Yaskawa INFORM job: SKRZYNIA_5040_0_STOPNI_1OBR.JBI

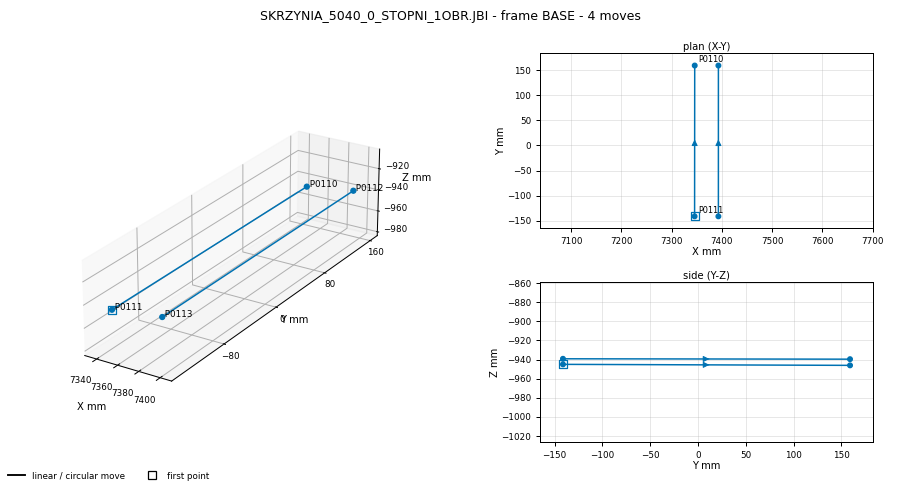
[picture p0: tool path of SKRZYNIA_5040_0_STOPNI_1OBR.JBI in frame BASE, 4 of 438 moves have a stored position in this frame; points joined in program order, loops and branches not executed]
/JOB
//NAME SKRZYNIA_5040_0_STOPNI_1OBR
///FOLDERNAME 02-SKRZYNIE_JOBS
//POS
///NPOS 514,514,0,47,4,0
///TOOL 0
///POSTYPE PULSE
///PULSE
C00000=1055,-24125,84372,288,19725,204
C00001=1055,-24125,84372,288,19725,204
C00002=25524,-25821,36823,19654,-58495,38520
C00003=23988,-24960,37134,18595,-57837,38812
C00004=22822,-23954,37534,17811,-57199,39017
C00005=22935,-24057,37491,17887,-57262,38997
C00006=20006,-24258,37408,15644,-56932,39751
C00007=24402,-25289,37013,18874,-58060,38740
C00008=22585,-24665,40358,17164,-59622,30036
C00009=23477,-23257,40205,18030,-58646,29630
C00010=22519,-22398,40568,17384,-58125,29795
C00011=22700,-22567,40495,17506,-58225,29764
C00012=19339,-22794,40398,14955,-57865,30607
C00013=24825,-24328,39798,18931,-59350,29401
C00014=0,-15438,65714,0,-68532,0
C00015=25524,-25821,36823,19654,-58495,38520
C00016=23988,-24960,37134,18595,-57837,38812
C00017=22822,-23954,37534,17811,-57199,39017
C00018=22935,-24057,37491,17887,-57262,38997
C00019=20006,-24258,37408,15644,-56932,39751
C00020=24402,-25289,37013,18874,-58060,38740
C00021=22585,-24665,40358,17164,-59622,30036
C00022=23477,-23257,40205,18030,-58646,29630
C00023=22519,-22398,40568,17384,-58125,29795
C00024=22700,-22567,40495,17506,-58225,29764
C00025=19339,-22794,40398,14955,-57865,30607
C00026=24825,-24328,39798,18931,-59350,29401
C00027=32755,-32613,25711,29640,-48730,33694
C00028=25632,-30899,26166,23992,-46203,35378
C00029=24264,-29862,26497,22996,-45413,35639
C00030=24403,-29974,26459,23097,-45496,35612
C00031=20575,-30233,26374,19602,-44891,36810
C00032=26556,-31526,25988,24663,-46720,35206
C00033=30846,-32795,25752,28021,-48338,30427
C00034=24953,-30697,26306,23444,-45946,31743
C00035=23937,-29910,26558,22702,-45353,31936
C00036=24039,-29993,26530,22778,-45414,31916
C00037=20322,-30240,26449,19379,-44834,33080
C00038=25997,-31433,26093,24205,-46535,31545
C00039=26028,-43665,26580,-39946,8682,24640
C00040=27956,-30595,53065,-101898,6609,54413
C00041=26028,-43663,26580,-39944,8677,24639
C00042=38784,-34544,25404,33956,-51320,34445
C00043=29266,-32676,25756,26732,-47889,36488
C00044=25734,-31262,26119,24020,-46377,37252
C00045=24289,-30200,26441,22967,-45549,37525
C00046=24367,-30262,26420,23025,-45594,37511
C00047=20043,-30544,26331,19080,-44922,38860
C00048=26573,-31816,25967,24631,-46839,37095
C00049=27817,-32566,25782,25532,-47502,36865
C00050=26896,-32020,25916,24865,-47014,37034
C00051=24344,-30243,26427,23007,-45578,37515
C00052=24432,-30312,26405,23072,-45630,37498
C00053=20021,-30599,26315,19050,-44944,38872
C00054=26262,-31616,26021,24405,-46667,37153
C00055=27439,-32346,25835,25259,-47302,36935
C00056=27343,-32252,25856,25196,-47233,36946
C00057=24581,-30384,26384,23190,-45695,37464
C00058=24689,-30466,26358,23269,-45758,37444
C00059=20001,-30771,26264,18999,-45026,38899
C00060=26308,-31607,26026,24448,-46671,37139
C00061=27526,-32360,25834,25329,-47326,36914
C00062=24269,-40076,6479,29767,-34177,34232
C00063=22958,-37632,10123,27061,-35370,35326
C00064=22703,-41294,1722,31272,-29953,33282
C00065=19440,-41515,1663,27208,-29122,34832
C00066=25465,-43501,1200,33269,-31905,32752
C00067=87177,-39066,-1236,81808,-72661,19198
C00068=4794,-34097,38974,4189,-31824,-1302
C00069=4794,-34097,38974,4189,13412,-1302
C00070=5394,-34032,37825,4779,8346,-1512
C00071=6591,-33902,35532,5956,-1761,-1932
C00072=10065,-33530,28876,9373,-31104,-3154
C00073=31877,-32319,25770,29025,-48287,33360
C00074=25247,-31158,26079,23631,-46177,35016
C00075=23652,-29939,26460,22464,-45250,35320
C00076=23742,-30013,26436,22530,-45305,35302
C00077=19630,-30281,26348,18756,-44677,36597
C00078=26056,-31710,25928,24219,-46631,34863
C00079=38095,-40136,7813,41252,-44156,24924
C00080=33231,-38681,8176,37792,-41757,25918
C00081=31538,-37640,8473,36716,-40716,26179
C00082=31687,-37737,8444,36811,-40809,26155
C00083=27389,-38154,8322,32773,-39589,27627
C00084=33834,-39023,8084,38175,-42120,25821
C00085=4264,-34194,25387,4006,-26954,-29436
C00086=4264,-34194,25387,4006,-26954,-81856
C00087=17634,-23800,39238,9573,-31425,-73339
C00088=17837,-27228,32238,10495,-29236,-73805
C00089=17837,-21535,44509,9322,-33342,-73155
C00090=17548,-20734,45666,8935,-33511,-73021
C00091=-20829,-18800,50532,-12466,-37179,-77446
C00092=-20884,-20901,46110,-12960,-35762,-77182
C00093=-20884,-26676,33664,-14451,-31668,-76336
C00094=-20624,-26699,33167,-14265,-31320,-76369
C00095=-33629,-40566,17444,-29603,-33447,-71192
C00096=-33629,-40566,17444,42578,-32312,-84654
C00097=-42160,-31266,16400,42578,-32312,-84654
C00098=-87798,-804,48829,-20188,-26072,-60966
C00099=-76454,-11934,10236,-25964,7954,-64922
C00100=-76448,-11928,10235,-25961,7944,-64914
C00101=-68643,-7759,-23318,-14097,50582,-74897
C00102=-70868,-8793,-8075,-29663,30364,-70765
C00103=-67243,-1968,12282,-49553,26687,-63567
C00104=-68655,-309,14069,-48513,25966,-64203
C00105=-67497,-1678,12591,-49367,26558,-63682
C00106=-71436,-723,2905,-26484,35140,-73726
C00107=-71436,176,6426,-27636,33595,-73066
C00108=-71434,778,8668,-28412,32633,-72624
C00109=-68624,-2689,-85,-28291,36551,-72622
C00110=-99375,3692,5712,40719,48607,-84097
C00111=-94964,4957,10918,40408,44640,-83792
C00112=-93063,6047,12199,39572,43744,-83178
C00113=-94964,4957,10918,40408,44640,-83792
C00114=-94964,5754,13918,41385,43553,-84439
C00115=-94964,4957,10918,40408,44640,-83792
C00116=-90271,-412,-5146,23417,46876,-76529
C00117=-83133,-4088,-8267,6704,41492,-71542
C00118=-83133,-4088,-8267,6704,41492,-71542
C00119=-83133,-4088,-8267,6704,41492,-11598
C00120=-83133,-16026,-8267,6704,41492,-11598
C00121=-83133,-16026,-8267,6704,41492,-11598
C00122=-48225,-19387,30619,3889,32460,-6728
C00123=56943,-39861,25115,1795,-37402,-69601
C00124=29960,-38386,-19607,-115769,-41858,-24264
C00125=65721,-6478,18155,-133323,-22195,3361
C00126=70544,4411,32968,-134868,-18623,4660
C00127=71874,8263,38598,-134556,-17327,4659
C00128=72629,9390,40002,-135279,-16924,5107
C00129=71441,7638,37831,-134139,-17555,4406
C00130=77146,8888,25050,-166574,-32612,18372
C00131=77146,10029,28643,-166204,-31014,18167
C00132=77146,11198,32202,-165803,-29459,17947
C00133=75508,4678,16951,-165715,-35157,17778
C00134=68680,12216,24468,-164340,-40455,-13359
C00135=68362,12845,25743,-164045,-40097,-13561
C00136=68362,13700,28585,-163752,-38808,-13742
C00137=68362,12845,25743,-164045,-40097,-13561
C00138=64993,-1168,28876,-102971,-10760,-49875
C00139=63888,481,30670,-102324,-11438,-50313
C00140=64993,-1168,28876,-102971,-10760,-49875
C00141=58588,-14653,4620,-120782,-19611,-35794
C00142=29960,-38386,-19607,-115769,-41858,-24264
C00143=56943,-39861,25115,1795,-37402,-69601
C00144=-1002,-39861,25115,1795,-37402,-69601
C00145=-1001,-39858,25114,1795,-37402,0
C00146=6591,-33902,35532,5956,-1761,-1932
C00147=6592,-33900,35531,103508,-35512,-26314
C00148=-99253,-13690,44082,59847,13407,-31313
C00149=-85045,-36869,-4353,28502,-22832,-52282
C00150=-92346,-18713,13565,21110,-22545,-55257
C00151=-85370,-14218,16934,32905,-23649,-60330
C00152=-84150,-13282,17685,34842,-23935,-61163
C00153=-82877,-12536,18624,36445,-24482,-61818
C00154=-84150,-13282,17685,34842,-23935,-61163
C00155=-85467,-11480,19558,33086,-23405,-60436
C00156=-84150,-13282,17685,34842,-23935,-61163
C00157=-85732,-21202,11427,30682,-24763,-59235
C00158=-84559,-15616,15722,33768,-24118,-60665
C00159=-84150,-13282,17685,34842,-23935,-61163
C00160=-83260,-12880,18034,36130,-24218,-61709
C00161=-84150,-13282,17685,34842,-23935,-61163
C00162=-85365,-11775,19006,33430,-23307,-60600
C00163=-84150,-13282,17685,34842,-23935,-61163
C00164=-85786,-16909,14677,31743,-23900,-59790
C00165=-84150,-13282,17685,34842,-23935,-61163
C00166=-83215,-12861,18051,36194,-24233,-61735
C00167=-84150,-13282,17685,34842,-23935,-61163
C00168=-85327,-11825,18959,33476,-23327,-60618
C00169=-84150,-13282,17685,34842,-23935,-61163
C00170=-87841,-18519,13420,28367,-23534,-58339
C00171=-84150,-13282,17685,34842,-23935,-61163
C00172=-83292,-12894,18020,36083,-24208,-61688
C00173=-84150,-13282,17685,34842,-23935,-61163
C00174=-85185,-12008,18799,33646,-23400,-60687
C00175=-84150,-13282,17685,34842,-23935,-61163
C00176=-86371,-18277,13606,30568,-23951,-59265
C00177=-84345,-13370,17612,34554,-23873,-61041
C00178=-83240,-12871,18042,36158,-24225,-61720
C00179=-84345,-13370,17612,34554,-23873,-61041
C00180=-85365,-12110,18711,33368,-23345,-60568
C00181=-84345,-13370,17612,34554,-23873,-61041
C00182=-86191,-19647,12567,30467,-24278,-59187
C00183=-84345,-13372,17610,34552,-23873,-61039
C00184=-83096,-12807,18098,36363,-24268,-61804
C00185=-84345,-13372,17610,34552,-23873,-61039
C00186=-85268,-12232,18600,33480,-23393,-60612
C00187=-84345,-13372,17610,34552,-23873,-61039
C00188=-84814,-16043,15376,33312,-24093,-60464
C00189=-84104,-13265,17702,34906,-23948,-61189
C00190=-82960,-12743,18153,36555,-24313,-61887
C00191=-84104,-13265,17702,34906,-23948,-61189
C00192=-84979,-12194,18635,33901,-23496,-60788
C00193=-84104,-13265,17702,34906,-23948,-61189
C00194=-86610,-16845,14732,30573,-23614,-59301
C00195=-84104,-13265,17702,34906,-23948,-61189
C00196=-82793,-12667,18222,36790,-24370,-61986
C00197=-84104,-13265,17702,34906,-23948,-61189
C00198=-84888,-12305,18537,34004,-23540,-60830
C00199=-84104,-13265,17702,34906,-23948,-61189
C00200=-83806,-19585,12613,33764,-25080,-60559
C00201=-83675,-13072,17868,35530,-24083,-61453
C00202=-82553,-12556,18319,37130,-24451,-62127
C00203=-83675,-13072,17868,35530,-24083,-61453
C00204=-84378,-12223,18610,34735,-23716,-61138
C00205=-83675,-13072,17868,35530,-24083,-61453
C00206=-87149,-17993,13826,29513,-23647,-58830
C00207=-84104,-13265,17702,34906,-23948,-61189
C00208=-82640,-12594,18285,37014,-24425,-62079
C00209=-84104,-13265,17702,34906,-23948,-61189
C00210=-84792,-12429,18430,34119,-23592,-60877
C00211=-84104,-13265,17702,34906,-23948,-61189
C00212=-83583,-9185,30892,23668,-36042,-57025
C00213=-85789,-8328,35795,20592,-37093,-55378
C00214=-85786,-16735,14816,31782,-23869,-59812
C00215=-84103,-13263,17702,34906,-23947,-61191
C00216=-83225,-12865,18046,36177,-24227,-61729
C00217=-84103,-13263,17702,34906,-23947,-61191
C00218=-84774,-12447,18412,34138,-23599,-60886
C00219=-84103,-13263,17702,34906,-23947,-61191
C00220=-86149,-16246,6730,18897,-35239,-57128
C00221=-86244,-15289,7532,18875,-35060,-57127
C00222=-85361,-14893,7870,19824,-35193,-57574
C00223=-86244,-15289,7532,18875,-35060,-57127
C00224=-86889,-14409,8282,18264,-34784,-56850
C00225=-86244,-15289,7532,18875,-35060,-57127
C00226=-90262,-21765,2389,14114,-35574,-54847
C00227=-90262,-21765,2389,28730,-17672,-54847
C00228=-89967,-19086,25635,28730,-17672,-54847
C00229=568,-24029,84339,168,19981,112
C00230=568,-24677,83015,164,20405,113
C00231=101153,-24598,83176,165,20353,113
C00232=101153,-24598,83176,165,20353,113
C00233=89967,-19086,25635,-28730,-17672,54847
C00234=90262,-21765,2389,-28730,-17672,54847
C00235=86932,-18662,4771,-17876,-35519,56628
C00236=86578,-15436,7408,-18515,-35011,56957
C00237=85428,-14922,7844,-19753,-35183,57541
C00238=84405,-14447,8250,-20842,-35348,58054
C00239=85428,-14922,7844,-19753,-35183,57541
C00240=86134,-13973,8661,-19091,-34881,57237
C00241=85428,-14922,7844,-19753,-35183,57541
C00242=85786,-16735,14816,-31782,-23869,59812
C00243=83514,-12996,17929,-35760,-24132,61552
C00244=82296,-12429,18424,-37488,-24534,62281
C00245=83514,-12996,17929,-35760,-24132,61552
C00246=84266,-12085,18725,-34910,-23738,61214
C00247=83514,-12996,17929,-35760,-24132,61552
C00248=87323,-6914,39851,-18853,-38149,44508
C00249=83118,-12818,18089,-36330,-24263,61791
C00250=81969,-12276,18566,-37944,-24648,62472
C00251=83118,-12818,18089,-36330,-24263,61791
C00252=83927,-11846,18941,-35423,-23842,61433
C00253=83118,-12818,18089,-36330,-24263,61791
C00254=83806,-19585,12613,-33764,-25080,60559
C00255=83148,-12832,18077,-36287,-24254,61773
C00256=81889,-12236,18598,-38058,-24676,62520
C00257=83148,-12832,18077,-36287,-24254,61773
C00258=83900,-11930,18867,-35446,-23862,61440
C00259=83148,-12832,18077,-36287,-24254,61773
C00260=86610,-16845,14732,-30573,-23614,59301
C00261=82493,-13239,17725,-37070,-24559,62089
C00262=81442,-12739,18159,-38529,-24915,62703
C00263=82493,-13239,17725,-37070,-24559,62089
C00264=83435,-12133,18689,-36040,-24063,61682
C00265=82493,-13239,17725,-37070,-24559,62089
C00266=84814,-16043,15376,-33312,-24093,60464
C00267=82555,-13613,17404,-36910,-24580,62015
C00268=81369,-13053,17885,-38558,-24979,62709
C00269=82555,-13613,17404,-36910,-24580,62015
C00270=83568,-12431,18429,-35805,-24046,61580
C00271=82555,-13613,17404,-36910,-24580,62015
C00272=86191,-19647,12567,-30467,-24278,59187
C00273=82500,-13648,17375,-36975,-24607,62039
C00274=81594,-13224,17740,-38236,-24911,62571
C00275=82500,-13648,17375,-36975,-24607,62039
C00276=83449,-12543,18332,-35941,-24104,61633
C00277=82500,-13648,17375,-36975,-24607,62039
C00278=86371,-18277,13606,-30568,-23951,59265
C00279=82904,-13790,17251,-36416,-24470,61808
C00280=81796,-13275,17692,-37971,-24838,62464
C00281=82904,-13790,17251,-36416,-24470,61808
C00282=83696,-12867,18046,-35547,-24051,61466
C00283=82904,-13790,17251,-36416,-24470,61808
C00284=87841,-18519,13420,-28367,-23534,58339
C00285=82748,-13879,17174,-36603,-24542,61883
C00286=81789,-13434,17554,-37946,-24861,62449
C00287=82748,-13879,17174,-36603,-24542,61883
C00288=83603,-12888,18026,-35668,-24086,61514
C00289=82748,-13879,17174,-36603,-24542,61883
C00290=85786,-16909,14677,-31743,-23900,59790
C00291=82339,-14116,16972,-37087,-24733,62079
C00292=81557,-13752,17280,-38171,-24994,62536
C00293=82339,-14116,16972,-37087,-24733,62079
C00294=83390,-12909,18006,-35951,-24172,61633
C00295=82339,-14116,16972,-37087,-24733,62079
C00296=85732,-21202,11427,-30682,-24763,59235
C00297=82398,-14365,16763,-36952,-24745,62014
C00298=81340,-13876,17176,-38416,-25096,62632
C00299=82398,-14365,16763,-36952,-24745,62014
C00300=83629,-12951,17972,-35620,-24090,61491
C00301=82398,-14365,16763,-36952,-24745,62014
C00302=92346,-18713,13565,-21110,-22545,55257
C00303=82794,-13980,17083,-36511,-24538,61844
C00304=81697,-13472,17516,-38043,-24902,62488
C00305=82794,-13980,17083,-36511,-24538,61844
C00306=83767,-12847,18056,-35444,-24023,61424
C00307=82794,-13980,17083,-36511,-24538,61844
C00308=85045,-36869,-4353,-28502,-22832,52282
C00309=69856,-53931,-13446,-33557,-28911,29591
C00310=73943,-28815,39553,-16801,-45089,19004
C00311=0,-24029,84339,0,19981,0
C00312=0,-24029,84339,0,19981,0
C00313=0,-52280,40443,0,6876,0
C00314=63961,-36661,14391,66570,-58199,13439
C00315=49610,-38907,493,64064,-47684,11073
C00316=46884,-37851,878,62974,-45995,11189
C00317=46721,-37909,857,62857,-45922,11231
C00318=54160,-39955,137,66075,-50361,10746
C00319=0,-52280,40443,0,6876,0
C00320=0,-52280,40443,0,6876,0
C00321=42978,-45587,7631,48214,-41849,18034
C00322=36694,-44945,-1657,49443,-34807,15750
C00323=45435,-38965,-3578,70378,-41546,11426
C00324=45248,-39111,-3491,69948,-41437,11613
C00325=32579,-45219,-13334,65473,-28542,22073
C00326=59828,-44646,-5405,72855,-48572,12139
C00327=0,-38761,66314,0,-763,0
C00328=0,-44757,54667,0,2744,0
C00329=40382,-38226,12225,48505,-40693,16039
C00330=55481,-27484,23768,62968,-54833,11978
C00331=49777,-26559,24206,59885,-51900,12566
C00332=49523,-31326,12270,55024,-55929,13117
C00333=55330,-33748,11238,57660,-59334,12681
C00334=78664,-24436,10378,82837,-79111,12029
C00335=75189,-23065,11287,81851,-76948,11927
C00336=75189,-45249,11287,81851,-38847,11927
C00337=29880,-45249,11287,43145,-11324,11927
C00338=0,-24029,84339,0,19981,0
C00339=0,-24026,84338,1,19977,2
C00340=4264,-34194,25387,4006,-26954,-29436
C00341=4264,-34194,25387,4006,-26954,-81856
C00342=18580,-28601,30698,11472,-29284,-74138
C00343=-23778,-26243,38799,-16502,-35132,-75964
C00344=18580,-28601,30698,11472,-29284,-74138
C00345=4264,-34194,25387,4006,-26954,-81856
C00346=4264,-34194,25387,4006,-26954,-29436
C00347=1,-24024,84337,2,19973,1
C00348=-64243,-26178,31107,-39513,40312,-5844
C00349=-72148,3973,56008,-35470,42045,-10522
C00350=-72090,16396,76301,-42067,35650,-6519
C00351=-69388,15725,61378,-31740,35177,-8719
C00352=-69127,27099,75569,-32744,34250,-8088
C00353=-67573,2495,11285,-21767,57629,-15193
C00354=-77819,19629,29798,-10454,63174,-20704
C00355=-72990,23583,14304,-10735,77209,-20379
C00356=-74593,38003,46707,-11043,65751,-19814
C00357=-73236,38943,48295,-11400,65557,-19316
C00358=-73329,42107,51779,-6346,67443,-19636
C00359=-87142,34654,46174,17622,63862,-25393
C00360=-87240,36727,48611,18897,66604,-25032
C00361=-99033,21517,12213,24947,79702,-26203
C00362=-91500,-14196,-34781,24472,81625,-22832
C00363=-100472,-45007,-27818,8167,67201,-29302
C00364=0,-36642,16905,0,48372,0
C00365=66009,-61997,-62105,21406,63483,18379
C00366=97242,-23579,-39442,10179,68876,30321
C00367=73684,-7073,-17511,24638,68131,29022
C00368=59136,7235,6676,33270,66602,27507
C00369=54816,14937,6234,39741,69494,31070
C00370=54365,20668,19279,41017,66202,29418
C00371=64503,4223,2857,29650,48528,26647
C00372=75622,3202,-3149,3890,49494,34281
C00373=88036,13177,2413,-18568,66573,35876
C00374=90462,21593,10123,-22613,76266,34479
C00375=92450,29224,20002,-25750,81642,33727
C00376=94949,8131,-12163,-20291,74229,36861
C00377=94949,8084,-13484,-20215,75047,36712
C00378=70412,-34016,-52305,-11724,65624,29757
C00379=44268,-30306,-1568,-7370,48673,18708
C00380=1,-24024,84337,2,19973,1
C00381=1,-24024,84337,2,19973,1
C00382=3796,-57671,22373,2336,-25309,-753
C00383=52632,-34554,16626,51161,-63050,5622
C00384=59461,-32779,9832,66317,-58406,17312
C00385=52772,-27880,19104,60329,-56577,14845
C00386=51509,-17404,41655,51674,-64690,19351
C00387=62932,-33588,12189,66848,-61063,18031
C00388=55769,-31640,17107,64026,-54372,11197
C00389=50117,-26891,23585,59871,-52280,12556
C00390=49716,-31387,12242,55119,-56039,13097
C00391=55330,-33748,11238,57660,-59334,12681
C00392=1,-24024,84337,2,19973,1
C00393=1,-24024,84337,2,19973,1
C00394=57188,-41777,19973,48132,-58706,4905
C00395=55566,-48748,-16991,79805,-45048,-6941
C00396=49908,-48716,-25784,90749,-41340,-3650
C00397=43896,-46926,-25352,90956,-37526,-4581
C00398=43530,-46832,-25319,90960,-37294,-4630
C00399=55479,-50244,-26473,91085,-44870,-3042
C00400=12119,-24859,71505,13236,4440,2633
C00401=-91085,-34291,10385,1908,-24348,-42097
C00402=-86191,-19647,12567,30467,-24278,-59187
C00403=-99288,-11708,19065,-14233,-20220,-40075
C00404=-98206,-11518,19604,-10142,-20308,-41629
C00405=-99474,-20389,12397,-11593,-22150,-41069
C00406=0,-52280,40443,0,6876,0
C00407=85348,-24204,23536,-13963,-15515,44275
C00408=84670,-17015,14597,-33277,-24304,60423
C00409=96971,-12584,18294,8365,-19955,42614
C00410=97182,-12918,18001,8747,-20027,42449
C00411=96230,-24528,9149,6144,-22576,43630
C00412=0,-52280,40443,0,6876,0
C00413=0,-52280,40443,0,6876,0
C00414=-90140,-60305,18108,-2708,1721,-7625
C00415=-95594,-27428,6866,-4663,-19832,-42154
C00416=-99356,-13410,18355,-15385,-17730,-37479
C00417=-99405,-10878,20508,-15853,-17333,-37255
C00418=-99132,-10804,20575,-15274,-17279,-37502
C00419=-99132,-3482,39129,-10940,-24351,-39674
C00420=-97546,-6584,14255,-163983,-14128,32873
C00421=-100183,-18601,14070,-16273,-18800,-37146
C00422=-90140,-60305,18108,-2708,1721,-7625
C00423=0,-52280,40443,0,6876,0
C00424=84259,-57935,27522,-3761,3673,6310
C00425=86507,-39672,4297,-27618,-16640,46340
C00426=70477,-27878,7073,-45786,-32339,64941
C00427=84043,-16293,15174,-34312,-24409,60872
C00428=100395,-12639,18246,19464,-20904,37830
C00429=99154,-17369,4403,32227,-9753,28926
C00430=99154,-17369,4403,32227,-9753,28926
C00431=98497,-14262,-10338,-9662,27059,46922
C00432=97745,-17327,14348,11122,-20983,41455
C00433=86507,-39672,4297,-27618,-16640,46340
C00434=84259,-57935,27522,-3761,3673,6310
C00435=0,-52280,40443,0,6876,0
C00436=0,-27933,77061,0,20812,0
C00437=0,-27933,77061,0,20812,0
C00438=0,-52280,40443,0,6876,0
C00439=-91970,-60791,14435,-3343,512,-9412
C00440=-99196,-15868,16098,-13748,-19297,-38710
C00441=-99196,-15868,16098,-13748,-19297,-38710
C00442=-99196,-15868,16098,-13748,-19297,-38710
C00443=-85815,-11758,19597,31748,-21097,-58265
C00444=-87383,-11883,19487,26986,-20206,-56250
C00445=-99562,-16264,15781,-14410,-19427,-38431
C00446=-99196,-15868,16098,-13748,-19297,-38710
C00447=-91970,-60791,14435,-3343,512,-9412
C00448=0,-52280,40443,0,6876,0
C00449=91083,-60784,14823,-9043,-825,15173
C00450=83869,-19403,12921,-33769,-24740,60260
C00451=83869,-19403,12921,-33769,-24740,60260
C00452=83420,-14897,16486,-35538,-24144,61113
C00453=90535,-11845,19652,-14037,-20800,51549
C00454=90317,-11662,19878,-14346,-20882,51648
C00455=95871,-14889,15992,4901,-19605,43825
C00456=83869,-19403,12921,-33769,-24740,60260
C00457=91083,-60784,14823,-9043,-825,15173
C00458=0,-52280,40443,0,6876,0
C00459=-91526,-60598,16699,7584,176,-13289
C00460=-94392,-6553,48683,5805,-47321,-49764
C00461=-88951,-345,54953,10686,-47392,-51569
C00462=-88172,5833,62122,11322,-47753,-51785
C00463=-90949,-14015,9500,8834,-34399,-51934
C00464=-84917,-15593,15742,33275,-23984,-60461
C00465=-81669,-15982,15425,37506,-25258,-62202
C00466=-79867,-25377,9541,37586,-25936,-59971
C00467=-91415,-60262,16631,7870,-73,-13734
C00468=24,-24029,84339,7,19981,5
C00469=160,-24029,84339,47,19981,32
C00470=99096,-24029,84339,47,19981,32
C00471=99096,-24029,84339,47,19981,32
C00472=89967,-19086,25635,-28730,-17672,54847
C00473=85786,-16735,14816,-31782,-23869,59812
C00474=83492,-14473,16674,-35480,-24338,61406
C00475=82628,-11567,19219,-37457,-24416,62267
C00476=85293,-13629,8874,-19696,-34851,57583
C00477=85505,-16299,6686,-19564,-35388,57437
C00478=89967,-19086,25635,-28730,-17672,54847
C00479=568,-24029,84339,168,19981,112
C00480=568,-24029,84339,168,19981,112
C00481=-91970,-60791,14435,-3343,512,-9412
C00482=-86948,-23217,10819,28314,-23349,-56438
C00483=-85895,-16522,15767,31843,-22281,-58087
C00484=-93643,1708,52973,2937,-38210,-34777
C00485=-93409,-737,47229,3345,-36106,-34967
C00486=-86145,-24679,9854,29028,-23971,-56682
C00487=-100471,-58311,4157,14142,-4822,-27614
C00488=-68517,-58311,4157,14142,-4822,-27614
C00489=0,-52280,40443,0,6876,0
C00490=91083,-60784,14823,-9043,-825,15173
C00491=83869,-19403,12921,-33769,-24740,60260
C00492=82620,-18743,14708,-32942,-26226,58979
C00493=83315,-11405,20766,-33572,-24860,59408
C00494=83326,-11144,20997,-33599,-24827,59423
C00495=84798,-22668,11879,-29033,-26372,57255
C00496=91083,-60784,14823,-9043,-825,15173
C00497=0,-52280,40443,0,6876,0
C00498=-6369,-39206,65423,-4801,-482,2563
C00499=-97287,-29142,12714,-8673,-22288,-37832
C00500=-86191,-19647,12567,30467,-24278,-59187
C00501=-85671,-16302,15857,30808,-24404,-58999
C00502=-99965,-10410,22406,-14600,-22538,-38834
C00503=-95758,-10871,21797,-1120,-21702,-44724
C00504=-87910,-17792,15835,25414,-24996,-56048
C00505=-97287,-29142,12714,-8673,-22288,-37832
C00506=0,-52280,40443,0,6876,0
C00507=92301,-25634,22749,2368,-15645,37646
C00508=83738,-18329,13570,-34202,-24868,60772
C00509=90096,-13099,18146,-15422,-20883,52700
C00510=93330,-13245,17928,-4627,-20146,48105
C00511=80226,-20465,12178,-39626,-27411,62762
C00512=92301,-25634,22749,2368,-15645,37646
C00513=0,-52280,40443,0,6876,0
BC00000=413138
BC00001=413138
BC00002=290246
BC00003=290246
BC00004=290246
BC00005=290246
BC00006=290246
BC00007=290246
BC00008=347127
BC00009=347132
BC00010=347132
BC00011=347132
BC00012=347132
BC00013=347132
BC00014=413138
BC00015=413134
BC00016=413134
BC00017=413134
BC00018=413134
BC00019=413134
BC00020=413134
BC00021=474623
BC00022=474628
BC00023=474628
BC00024=474628
BC00025=474628
BC00026=474628
BC00027=522849
BC00028=522849
BC00029=522849
BC00030=522849
BC00031=522849
BC00032=522849
BC00033=586045
BC00034=586045
BC00035=586045
BC00036=586045
BC00037=586045
BC00038=586045
BC00039=479622
BC00040=618860
BC00041=673957
BC00042=655410
BC00043=655410
BC00044=655410
BC00045=655410
BC00046=655410
BC00047=655410
BC00048=655410
BC00049=708270
BC00050=708270
BC00051=708270
BC00052=708270
BC00053=708270
BC00054=708270
BC00055=770184
BC00056=770184
BC00057=770184
BC00058=770184
BC00059=770184
BC00060=770184
BC00061=823730
BC00062=829967
BC00063=829969
BC00064=829970
BC00065=829970
BC00066=829970
BC00067=838761
BC00068=740349
BC00069=687700
BC00070=771943
BC00071=861898
BC00072=881669
BC00073=901229
BC00074=901229
BC00075=901229
BC00076=901229
BC00077=901229
BC00078=901229
BC00079=949836
BC00080=949836
BC00081=949836
BC00082=949836
BC00083=949836
BC00084=949836
BC00085=926513
BC00086=926513
BC00087=911152
BC00088=911152
BC00089=915598
BC00090=915598
BC00091=915598
BC00092=915598
BC00093=915598
BC00094=915598
BC00095=915598
BC00096=915598
BC00097=915598
BC00098=915598
BC00099=915598
BC00100=933350
BC00101=944436
BC00102=961140
BC00103=961140
BC00104=961140
BC00105=961140
BC00106=961140
BC00107=961140
BC00108=961141
BC00109=961141
BC00110=961141
BC00111=961141
BC00112=961141
BC00113=961141
BC00114=961141
BC00115=961141
BC00116=951518
BC00117=936884
BC00118=911619
BC00119=911619
BC00120=911619
BC00121=878437
BC00122=844004
BC00123=915598
BC00124=915598
BC00125=915598
BC00126=931812
BC00127=936973
BC00128=936973
BC00129=936973
BC00130=936973
BC00131=936973
BC00132=936973
BC00133=936973
BC00134=936973
BC00135=936973
BC00136=936973
BC00137=936973
BC00138=936973
BC00139=936973
BC00140=936973
BC00141=931460
BC00142=915598
BC00143=915598
BC00144=915598
BC00145=930961
BC00146=861898
BC00147=861901
BC00148=861901
BC00149=931504
BC00150=963634
BC00151=963631
BC00152=963631
BC00153=963631
BC00154=963631
BC00155=963631
BC00156=963631
BC00157=902188
BC00158=902188
BC00159=902188
BC00160=902188
BC00161=902188
BC00162=902188
BC00163=902188
BC00164=840744
BC00165=840744
BC00166=840744
BC00167=840744
BC00168=840744
BC00169=840744
BC00170=779300
BC00171=779300
BC00172=779300
BC00173=779300
BC00174=779300
BC00175=779300
BC00176=717855
BC00177=717855
BC00178=717855
BC00179=717855
BC00180=717855
BC00181=717855
BC00182=656405
BC00183=656405
BC00184=656405
BC00185=656405
BC00186=656405
BC00187=656405
BC00188=594961
BC00189=594961
BC00190=594961
BC00191=594961
BC00192=594961
BC00193=594961
BC00194=533517
BC00195=533517
BC00196=533517
BC00197=533517
BC00198=533517
BC00199=533517
BC00200=472073
BC00201=472073
BC00202=472073
BC00203=472073
BC00204=472073
BC00205=472073
BC00206=410629
BC00207=410629
BC00208=410629
BC00209=410629
BC00210=410629
BC00211=410629
BC00212=410629
BC00213=349186
BC00214=349186
BC00215=349186
BC00216=349186
BC00217=349186
BC00218=349186
BC00219=349186
BC00220=336469
BC00221=336469
BC00222=336469
BC00223=336469
BC00224=336469
BC00225=336469
BC00226=336469
BC00227=336469
BC00228=336469
BC00229=336469
BC00230=511557
BC00231=512005
BC00232=363797
BC00233=336469
BC00234=336469
BC00235=337415
BC00236=337415
BC00237=337415
BC00238=337415
BC00239=337415
BC00240=337415
BC00241=337415
BC00242=349186
BC00243=350137
BC00244=350137
BC00245=350137
BC00246=350137
BC00247=350137
BC00248=410629
BC00249=411580
BC00250=411580
BC00251=411580
BC00252=411580
BC00253=411580
BC00254=472073
BC00255=473025
BC00256=473025
BC00257=473025
BC00258=473025
BC00259=473025
BC00260=533517
BC00261=534468
BC00262=534468
BC00263=534468
BC00264=534468
BC00265=534468
BC00266=594961
BC00267=594961
BC00268=594961
BC00269=594961
BC00270=594961
BC00271=594961
BC00272=656405
BC00273=657350
BC00274=657350
BC00275=657350
BC00276=657350
BC00277=657350
BC00278=717855
BC00279=718799
BC00280=718799
BC00281=718799
BC00282=718799
BC00283=718799
BC00284=779300
BC00285=780245
BC00286=780245
BC00287=780245
BC00288=780245
BC00289=780245
BC00290=840744
BC00291=841691
BC00292=841691
BC00293=841691
BC00294=841691
BC00295=841691
BC00296=902188
BC00297=903136
BC00298=903136
BC00299=903136
BC00300=903136
BC00301=903136
BC00302=963634
BC00303=963633
BC00304=963633
BC00305=963633
BC00306=963633
BC00307=963633
BC00308=931504
BC00309=861901
BC00310=861901
BC00311=769966
BC00312=769966
BC00313=716865
BC00314=660977
BC00315=660977
BC00316=660977
BC00317=717171
BC00318=717171
BC00319=716865
BC00320=796033
BC00321=895097
BC00322=895097
BC00323=895097
BC00324=945882
BC00325=955598
BC00326=945882
BC00327=840120
BC00328=538973
BC00329=485226
BC00330=456696
BC00331=456696
BC00332=417276
BC00333=417276
BC00334=493986
BC00335=514306
BC00336=514306
BC00337=514306
BC00338=493986
BC00339=797003
BC00340=895791
BC00341=895791
BC00342=895791
BC00343=900237
BC00344=895791
BC00345=895791
BC00346=895791
BC00347=766279
BC00348=781641
BC00349=781641
BC00350=838351
BC00351=858237
BC00352=883176
BC00353=915108
BC00354=915108
BC00355=942617
BC00356=942617
BC00357=942617
BC00358=942618
BC00359=942618
BC00360=942619
BC00361=942619
BC00362=942619
BC00363=857277
BC00364=815875
BC00365=899415
BC00366=938535
BC00367=938536
BC00368=938536
BC00369=968783
BC00370=968783
BC00371=968783
BC00372=968783
BC00373=968783
BC00374=968786
BC00375=968786
BC00376=968786
BC00377=942380
BC00378=942380
BC00379=873567
BC00380=781640
BC00381=476651
BC00382=522561
BC00383=566531
BC00384=593948
BC00385=593948
BC00386=529848
BC00387=529848
BC00388=333808
BC00389=332068
BC00390=295166
BC00391=294388
BC00392=461290
BC00393=663315
BC00394=778314
BC00395=778312
BC00396=778312
BC00397=778312
BC00398=838222
BC00399=838222
BC00400=566410
BC00401=679663
BC00402=656405
BC00403=656405
BC00404=717855
BC00405=717855
BC00406=717855
BC00407=662303
BC00408=657350
BC00409=657350
BC00410=718803
BC00411=718803
BC00412=717855
BC00413=792672
BC00414=792672
BC00415=896850
BC00416=895720
BC00417=895720
BC00418=957178
BC00419=957178
BC00420=957178
BC00421=957178
BC00422=792672
BC00423=792672
BC00424=792672
BC00425=887446
BC00426=903126
BC00427=903126
BC00428=903126
BC00429=964577
BC00430=976097
BC00431=976097
BC00432=964577
BC00433=887446
BC00434=792672
BC00435=792672
BC00436=700249
BC00437=546214
BC00438=546214
BC00439=546211
BC00440=546211
BC00441=406776
BC00442=406776
BC00443=406778
BC00444=468200
BC00445=468200
BC00446=546211
BC00447=546211
BC00448=546214
BC00449=546214
BC00450=507604
BC00451=410782
BC00452=410782
BC00453=410782
BC00454=472720
BC00455=472720
BC00456=507604
BC00457=546214
BC00458=546214
BC00459=516757
BC00460=383716
BC00461=349186
BC00462=349186
BC00463=336469
BC00464=349186
BC00465=410629
BC00466=416512
BC00467=515801
BC00468=520018
BC00469=474013
BC00470=474013
BC00471=403108
BC00472=336469
BC00473=349186
BC00474=349186
BC00475=349186
BC00476=337415
BC00477=337415
BC00478=336469
BC00479=336469
BC00480=428401
BC00481=546211
BC00482=591088
BC00483=591088
BC00484=591088
BC00485=531116
BC00486=529640
BC00487=529640
BC00488=529640
BC00489=529640
BC00490=546214
BC00491=589919
BC00492=595627
BC00493=595627
BC00494=534177
BC00495=534177
BC00496=546214
BC00497=529640
BC00498=651195
BC00499=765890
BC00500=777968
BC00501=778453
BC00502=779252
BC00503=840748
BC00504=840748
BC00505=765890
BC00506=717855
BC00507=741100
BC00508=780224
BC00509=780222
BC00510=841743
BC00511=841743
BC00512=741100
BC00513=717855
///POSTYPE BASE
///RECTAN
///RCONF 1,0,0,0,0,0,0,0,0,0,0,0,0,0,0,0,0,0,0,0,0,0,0,0
P00006=-0.171,0.002,6.340,0.0000,0.0000,0.0000
///RCONF 0,0,0,0,0,0,0,0,0,0,0,0,0,0,0,0,0,0,0,0,0,0,0,0
P00021=6.550,-0.003,-5.735,0.0000,0.0000,0.0000
P00023=7.025,-0.019,-7.168,0.0000,0.0000,0.0000
///RCONF 1,0,0,0,0,0,0,0,0,0,0,0,0,0,0,0,0,0,0,0,0,0,0,0
P00098=-0.089,-2.467,4.059,0.0000,0.0000,0.0000
P00099=0.011,-2.380,1.226,0.0000,0.0000,0.0000
P00100=-0.081,2.558,4.482,0.0000,0.0000,0.0000
P00101=0.030,-2.286,2.993,0.0000,0.0000,0.0000
P00102=-0.005,-1.108,1.644,0.0000,0.0000,0.0000
P00103=-0.094,-3.400,4.200,0.0000,0.0000,0.0000
P00104=0.043,-2.127,5.826,0.0000,0.0000,0.0000
P00105=-0.043,0.662,5.286,0.0000,0.0000,0.0000
P00106=-0.018,-2.519,0.237,0.0000,0.0000,0.0000
P00107=-0.008,-4.537,-4.500,0.0000,0.0000,0.0000
P00108=0.014,-3.040,2.637,0.0000,0.0000,0.0000
P00109=0.017,-3.622,2.341,0.0000,0.0000,0.0000
P00110=7346.140,158.997,-946.107,-0.1876,37.7131,-155.1643
P00111=7345.905,-141.160,-945.062,8.1413,34.2244,-174.1788
P00112=7393.287,158.977,-939.640,-0.1938,37.7128,-155.1905
P00113=7393.259,-141.170,-939.228,8.1507,34.2195,-174.1496
///RCONF 0,0,0,0,0,0,0,0,0,0,0,0,0,0,0,0,0,0,0,0,0,0,0,0
P00280=-0.761,-1.221,0.004,0.0000,0.0000,0.0000
///RCONF 1,0,0,0,0,0,0,0,0,0,0,0,0,0,0,0,0,0,0,0,0,0,0,0
P00281=-0.866,-3.587,-0.008,0.0000,0.0000,0.0000
///RCONF 0,0,0,0,1,0,0,0,0,0,0,0,0,0,0,0,0,0,0,0,0,0,0,0
P00290=-0.023,-0.050,5.560,0.0000,0.0000,0.0000
///RCONF 1,0,0,0,0,0,0,0,0,0,0,0,0,0,0,0,0,0,0,0,0,0,0,0
P00291=0.002,-0.893,4.526,0.0000,0.0000,0.0000
P00300=-0.036,-1.505,2.318,0.0000,0.0000,0.0000
P00301=0.046,-2.112,7.779,0.0000,0.0000,0.0000
P00302=-0.171,0.002,6.340,0.0000,0.0000,0.0000
///RCONF 0,0,0,0,0,0,0,0,0,0,0,0,0,0,0,0,0,0,0,0,0,0,0,0
P00303=-0.004,-1.437,-4.584,0.0000,0.0000,0.0000
P00304=0.028,-1.666,-4.234,0.0000,0.0000,0.0000
P00305=-0.003,-1.920,-3.501,0.0000,0.0000,0.0000
P00306=0.015,-2.252,-3.054,0.0000,0.0000,0.0000
P00307=0.019,-2.151,-5.077,0.0000,0.0000,0.0000
P00308=-0.003,-2.092,-4.888,0.0000,0.0000,0.0000
P00309=-0.040,-2.205,-4.992,0.0000,0.0000,0.0000
P00310=-0.006,-2.490,-5.925,0.0000,0.0000,0.0000
P00311=-0.007,-2.079,-5.307,0.0000,0.0000,0.0000
P00350=11.519,-0.008,1.149,0.0000,0.0000,0.0000
P00351=13.563,-0.027,-0.653,0.0000,0.0000,0.0000
P00352=13.252,-0.027,-0.827,0.0000,0.0000,0.0000
P00353=10.971,-0.082,0.776,0.0000,0.0000,0.0000
P00354=-0.024,2.508,-1.824,0.0000,0.0000,0.0000
P00355=-0.001,2.528,-1.131,0.0000,0.0000,0.0000
P00356=-0.034,2.921,-0.262,0.0000,0.0000,0.0000
P00357=0.003,3.386,-0.091,0.0000,0.0000,0.0000
P00358=0.014,3.037,-0.020,0.0000,0.0000,0.0000
P00359=-0.005,2.731,0.912,0.0000,0.0000,0.0000
P00360=-0.011,3.412,0.438,0.0000,0.0000,0.0000
P00361=0.018,3.050,1.253,0.0000,0.0000,0.0000
BP00110=5931.608
BP00111=5960.552
BP00112=5960.545
BP00113=5960.552
//INST
///DATE 2025/03/18 15:47
///ATTR SC,RW
///GROUP1 RB1,BS1
NOP
CALL JOB:MOVE_INTO_TUNNEL
MOVJ C00000 BC00000 VJ=30.00
'------------------------
'------------------------
'SPOINA SRODEK DOL
'------------------------
'------------------------
'POMIAR DO WYJ!! PRZEROBIC NA STD
MOVJ C00001 BC00001 VJ=40.00
'SPOINA_PODLOGA_BRAK_ROZP
MOVJ C00002 BC00002 VJ=20.00 PL=0
MOVL C00003 BC00003 V=166.7 PL=0
REFP 3 C00004 BC00004
CALL JOB:SEARCH-R1
SET P0098 P0006
SFTON P0098
MOVL C00005 BC00005 V=66.7 PL=0
REFP 3 C00006 BC00006
CALL JOB:SEARCH-R1
SET P0098 P0006
SFTON P0098
MOVL C00007 BC00007 V=333.3 PL=0
SFTOF
'W3L
MOVL C00008 BC00008 V=666.7
MOVL C00009 BC00009 V=166.7 PL=0
REFP 3 C00010 BC00010
CALL JOB:SEARCH-R1
SET P0099 P0006
SFTON P0099
MOVL C00011 BC00011 V=166.7 PL=0
REFP 3 C00012 BC00012
CALL JOB:SEARCH-R1
SET P0099 P0006
SFTON P0099
MOVL C00013 BC00013 V=333.3 PL=0
SFTOF
'SPOINA_PODLOGA_BRAK_ROZP
MOVJ C00014 BC00014 VJ=40.00
'W3P
MOVJ C00015 BC00015 VJ=20.00 PL=0
MOVL C00016 BC00016 V=166.7 PL=0
REFP 3 C00017 BC00017
CALL JOB:SEARCH-R1
SET P0100 P0006
SFTON P0100
MOVL C00018 BC00018 V=66.7 PL=0
REFP 3 C00019 BC00019
CALL JOB:SEARCH-R1
SET P0100 P0006
SFTON P0100
MOVL C00020 BC00020 V=333.3 PL=0
SFTOF
'W3L
MOVL C00021 BC00021 V=666.7
MOVL C00022 BC00022 V=166.7 PL=0
REFP 3 C00023 BC00023
CALL JOB:SEARCH-R1
SET P0101 P0006
SFTON P0101
MOVL C00024 BC00024 V=166.7 PL=0
REFP 3 C00025 BC00025
CALL JOB:SEARCH-R1
SET P0101 P0006
SFTON P0101
MOVL C00026 BC00026 V=333.3 PL=0
SFTOF
'W9P
MOVL C00027 BC00027 V=666.7
MOVL C00028 BC00028 V=166.7
REFP 3 C00029 BC00029
CALL JOB:SEARCH-R1
SET P0102 P0006
SFTON P0102
MOVL C00030 BC00030 V=166.7 PL=0
REFP 3 C00031 BC00031
CALL JOB:SEARCH-R1
SET P0102 P0006
SFTON P0102
MOVL C00032 BC00032 V=333.3 PL=0
'W9L
MOVL C00033 BC00033 V=666.7
MOVL C00034 BC00034 V=166.7
REFP 3 C00035 BC00035
CALL JOB:SEARCH-R1
SET P0103 P0006
SFTON P0103
MOVL C00036 BC00036 V=166.7 PL=0
REFP 3 C00037 BC00037
CALL JOB:SEARCH-R1
SET P0103 P0006
SFTON P0103
MOVL C00038 BC00038 V=333.3 PL=0
'PRZEJAZ NAD BELKA
MOVL C00039 BC00039 V=666.7
MOVJ C00040 BC00040 VJ=40.00
MOVJ C00041 BC00041 VJ=40.00
MOVJ C00042 BC00042 VJ=40.00
'W1P
MOVJ C00043 BC00043 VJ=20.00 PL=0
MOVL C00044 BC00044 V=166.7 PL=0
REFP 3 C00045 BC00045
CALL JOB:SEARCH-R1
SET P0104 P0006
SFTON P0104
MOVL C00046 BC00046 V=166.7 PL=0
REFP 3 C00047 BC00047
CALL JOB:SEARCH-R1
SET P0104 P0006
SFTON P0104
MOVL C00048 BC00048 V=333.3 PL=0
SFTOF
'W1L
MOVL C00049 BC00049 V=666.7
MOVL C00050 BC00050 V=166.7 PL=0
REFP 3 C00051 BC00051
CALL JOB:SEARCH-R1
SET P0105 P0006
SFTON P0105
MOVL C00052 BC00052 V=166.7 PL=0
REFP 3 C00053 BC00053
CALL JOB:SEARCH-R1
SET P0105 P0006
SFTON P0105
MOVL C00054 BC00054 V=333.3 PL=0
SFTOF
MOVL C00055 BC00055 V=666.7
'W10P
MOVL C00056 BC00056 V=166.7 PL=0
REFP 3 C00057 BC00057
CALL JOB:SEARCH-R1
SET P0106 P0006
SFTON P0106
MOVL C00058 BC00058 V=166.7 PL=0
REFP 3 C00059 BC00059
CALL JOB:SEARCH-R1
SET P0106 P0006
SFTON P0106
MOVL C00060 BC00060 V=333.3 PL=0
SFTOF
'W10L
MOVL C00061 BC00061 V=333.3
MOVL C00062 BC00062 V=166.7 PL=0
REFP 3 C00063 BC00063
CALL JOB:SEARCH-R1
SET P0107 P0006
SFTON P0107
MOVL C00064 BC00064 V=166.7 PL=0
REFP 3 C00065 BC00065
CALL JOB:SEARCH-R1
SET P0107 P0006
SFTON P0107
MOVL C00066 BC00066 V=333.3 PL=0
SFTOF
MOVL C00067 BC00067 V=333.3
'PRZEJAZD
MOVJ C00068 BC00068 VJ=50.00
MOVJ C00069 BC00069 VJ=50.00
MOVJ C00070 BC00070 VJ=60.00
MOVJ C00071 BC00071 VJ=60.00
MOVJ C00072 BC00072 VJ=60.00
MOVJ C00073 BC00073 VJ=60.00 PL=0
MOVL C00074 BC00074 V=166.7 PL=0
REFP 3 C00075 BC00075
CALL JOB:SEARCH-R1
SET P0108 P0006
SFTON P0108
MOVL C00076 BC00076 V=166.7 PL=0
REFP 3 C00077 BC00077
CALL JOB:SEARCH-R1
SET P0108 P0006
SFTON P0108
MOVL C00078 BC00078 V=333.3 PL=0
SFTOF
'W2P
'W2L
MOVL C00079 BC00079 V=666.7
MOVL C00080 BC00080 V=166.7 PL=0
REFP 3 C00081 BC00081
CALL JOB:SEARCH-R1
SET P0109 P0006
SFTON P0109
MOVL C00082 BC00082 V=166.7 PL=0
REFP 3 C00083 BC00083
CALL JOB:SEARCH-R1
SET P0109 P0006
SFTON P0109
MOVL C00084 BC00084 V=333.3 PL=0
SFTOF
'PRZEJAZD
'POMIAR DO WYJ!! PRZEROBIC NA STD
'KONIEC
MOVJ C00085 BC00085 VJ=40.00
MOVJ C00086 BC00086 VJ=50.00
'W5L
MOVJ C00087 BC00087 VJ=30.00 PL=0
SET I020 110
CALL JOB:SEARCH_Z-40_Z1_X40
MOVL C00088 BC00088 V=166.7
'W6L
MOVJ C00089 BC00089 VJ=20.00 PL=0
SET I020 112
CALL JOB:SEARCH_Z-40_Z1_X40
MOVL C00090 BC00090 V=166.7
'W6P
MOVL C00091 BC00091 V=150.0 PL=0
SET I020 113
CALL JOB:SEARCH_Z-40_Z1_X40
MOVL C00092 BC00092 V=166.7
'W5P
MOVJ C00093 BC00093 VJ=20.00 PL=0
SET I020 111
CALL JOB:SEARCH_Z-40_Z1_X40
MOVL C00094 BC00094 V=166.7
'W7A
MOVJ C00095 BC00095 VJ=40.00
MOVJ C00096 BC00096 VJ=40.00
MOVJ C00097 BC00097 VJ=40.00
MOVJ C00098 BC00098 VJ=40.00
MOVJ C00099 BC00099 VJ=40.00
MOVJ C00100 BC00100 VJ=40.00
MOVJ C00101 BC00101 VJ=40.00
MOVJ C00102 BC00102 VJ=40.00
MOVL C00103 BC00103 V=250.0
REFP 3 C00104 BC00104
CALL JOB:SEARCH-R1
SET P0280 P0006
SFTON P0280
MOVL C00105 BC00105 V=166.7
MOVL C00106 BC00106 V=250.0
MOVL C00107 BC00107 V=166.7
REFP 3 C00108 BC00108
CALL JOB:SEARCH-R1
SET P0280 P0006
MOVL C00109 BC00109 V=166.7
SFTOF
MOVL C00110 BC00110 V=333.3
MOVL C00111 BC00111 V=166.7
REFP 3 C00112 BC00112
CALL JOB:SEARCH-R1
SET P0290 P0006
SFTON P0290
MOVL C00113 BC00113 V=166.7
REFP 3 C00114 BC00114
CALL JOB:SEARCH-R1
SET P0290 P0006
MOVL C00115 BC00115 V=166.7
'DOKONCZYC SEARCH
'DOKONCZYC SEARCH
MOVJ C00116 BC00116 VJ=20.00
SFTOF
MOVJ C00117 BC00117 VJ=30.00
MOVJ C00118 BC00118 VJ=40.00
MOVJ C00119 BC00119 VJ=40.00
MOVJ C00120 BC00120 VJ=40.00
MOVJ C00121 BC00121 VJ=40.00
MOVJ C00122 BC00122 VJ=50.00
'W7B
MOVJ C00123 BC00123 VJ=50.00
MOVJ C00124 BC00124 VJ=50.00
MOVJ C00125 BC00125 VJ=30.00
MOVJ C00126 BC00126 VJ=20.00
MOVL C00127 BC00127 V=166.7
REFP 3 C00128 BC00128
CALL JOB:SEARCH-R1
SET P0281 P0006
MOVL C00129 BC00129 V=166.7
SFTON P0281
MOVL C00130 BC00130 V=166.7
MOVL C00131 BC00131 V=166.7
REFP 3 C00132 BC00132
CALL JOB:SEARCH-R1
SET P0281 P0006
MOVJ C00133 BC00133 VJ=15.00
SFTOF
MOVJ C00134 BC00134 VJ=20.00
MOVL C00135 BC00135 V=166.7
REFP 3 C00136 BC00136
CALL JOB:SEARCH-R1
SET P0291 P0006
MOVL C00137 BC00137 V=166.7
MOVL C00138 BC00138 V=166.7
REFP 3 C00139 BC00139
CALL JOB:SEARCH-R1
SET P0291 P0006
MOVL C00140 BC00140 V=166.7
'DOKONCZYC SEARCH
'DOKONCZYC SEARCH
'DOKONCZYC SEARCH
MOVJ C00141 BC00141 VJ=30.00
MOVJ C00142 BC00142 VJ=30.00
MOVJ C00143 BC00143 VJ=50.00
MOVJ C00144 BC00144 VJ=50.00
'------------------------
'------------------------
'PRAWA STRONA PROFIL GORA
'------------------------
'------------------------
MOVJ C00145 BC00145 VJ=50.00
MOVJ C00146 BC00146 VJ=50.00
MOVJ C00147 BC00147 VJ=50.00
MOVJ C00148 BC00148 VJ=20.00
MOVJ C00149 BC00149 VJ=50.00
'------------------------
'W14A L
'------------------------
SFTOF
MOVJ C00150 BC00150 VJ=50.00
MOVJ C00151 BC00151 VJ=30.00
MOVL C00152 BC00152 V=166.7 PL=0
REFP 3 C00153 BC00153
CALL JOB:SEARCH-R1
SET P0300 P0006
SFTON P0300
MOVL C00154 BC00154 V=166.7 PL=0
REFP 3 C00155 BC00155
CALL JOB:SEARCH-R1
SET P0300 P0006
SFTON P0300
MOVL C00156 BC00156 V=166.7 PL=0
SFTOF
'------------------------
'W14A P
'------------------------
SFTOF
MOVJ C00157 BC00157 VJ=50.00
MOVJ C00158 BC00158 VJ=50.00
MOVL C00159 BC00159 V=166.7 PL=0
REFP 3 C00160 BC00160
CALL JOB:SEARCH-R1
SET P0301 P0006
SFTON P0301
MOVL C00161 BC00161 V=166.7 PL=0
REFP 3 C00162 BC00162
CALL JOB:SEARCH-R1
SET P0301 P0006
SFTON P0301
MOVL C00163 BC00163 V=166.7 PL=0
SFTOF
'------------------------
'W19A L
'------------------------
SFTOF
MOVJ C00164 BC00164 VJ=50.00
MOVL C00165 BC00165 V=200.0 PL=0
REFP 3 C00166 BC00166
CALL JOB:SEARCH-R1
SET P0302 P0006
SFTON P0302
MOVL C00167 BC00167 V=166.7 PL=0
REFP 3 C00168 BC00168
CALL JOB:SEARCH-R1
SET P0302 P0006
SFTON P0302
MOVL C00169 BC00169 V=250.0 PL=0
SFTOF
'------------------------
'W19A P
'------------------------
SFTOF
MOVJ C00170 BC00170 VJ=50.00
MOVL C00171 BC00171 V=166.7 PL=0
REFP 3 C00172 BC00172
CALL JOB:SEARCH-R1
SET P0303 P0006
SFTON P0303
MOVL C00173 BC00173 V=166.7 PL=0
REFP 3 C00174 BC00174
CALL JOB:SEARCH-R1
SET P0303 P0006
SFTON P0303
MOVL C00175 BC00175 V=166.7 PL=0
SFTOF
'------------------------
'W13A L
'------------------------
SFTOF
MOVJ C00176 BC00176 VJ=50.00
MOVL C00177 BC00177 V=166.7 PL=0
REFP 3 C00178 BC00178
CALL JOB:SEARCH-R1
SET P0304 P0006
SFTON P0304
MOVL C00179 BC00179 V=166.7 PL=0
REFP 3 C00180 BC00180
CALL JOB:SEARCH-R1
SET P0304 P0006
SFTON P0304
MOVL C00181 BC00181 V=166.7 PL=0
SFTOF
'------------------------
'W13A P
'------------------------
SFTOF
MOVJ C00182 BC00182 VJ=50.00
MOVL C00183 BC00183 V=200.0 PL=0
REFP 3 C00184 BC00184
CALL JOB:SEARCH-R1
SET P0305 P0006
SFTON P0305
MOVL C00185 BC00185 V=166.7 PL=0
REFP 3 C00186 BC00186
CALL JOB:SEARCH-R1
SET P0305 P0006
SFTON P0305
MOVL C00187 BC00187 V=250.0 PL=0
SFTOF
'------------------------
'W18A L
'------------------------
SFTOF
MOVJ C00188 BC00188 VJ=50.00
MOVL C00189 BC00189 V=200.0 PL=0
REFP 3 C00190 BC00190
CALL JOB:SEARCH-R1
SET P0306 P0006
SFTON P0306
MOVL C00191 BC00191 V=166.7 PL=0
REFP 3 C00192 BC00192
CALL JOB:SEARCH-R1
SET P0306 P0006
SFTON P0306
MOVL C00193 BC00193 V=166.7 PL=0
SFTOF
'------------------------
'W18A P
'------------------------
SFTOF
MOVJ C00194 BC00194 VJ=50.00
MOVL C00195 BC00195 V=200.0 PL=0
REFP 3 C00196 BC00196
CALL JOB:SEARCH-R1
SET P0307 P0006
SFTON P0307
MOVL C00197 BC00197 V=166.7 PL=0
REFP 3 C00198 BC00198
CALL JOB:SEARCH-R1
SET P0307 P0006
SFTON P0307
MOVL C00199 BC00199 V=166.7 PL=0
SFTOF
'------------------------
'W15A L
'------------------------
SFTOF
MOVJ C00200 BC00200 VJ=50.00
MOVL C00201 BC00201 V=200.0 PL=0
REFP 3 C00202 BC00202
CALL JOB:SEARCH-R1
SET P0308 P0006
SFTON P0308
MOVL C00203 BC00203 V=166.7 PL=0
REFP 3 C00204 BC00204
CALL JOB:SEARCH-R1
SET P0308 P0006
SFTON P0308
MOVL C00205 BC00205 V=166.7 PL=0
SFTOF
'------------------------
'W15A P
'------------------------
SFTOF
MOVJ C00206 BC00206 VJ=50.00
MOVL C00207 BC00207 V=166.7 PL=0
REFP 3 C00208 BC00208
CALL JOB:SEARCH-R1
SET P0309 P0006
SFTON P0309
MOVL C00209 BC00209 V=166.7 PL=0
REFP 3 C00210 BC00210
CALL JOB:SEARCH-R1
SET P0309 P0006
SFTON P0309
MOVL C00211 BC00211 V=166.7 PL=0
SFTOF
MOVL C00212 BC00212 V=333.3
'------------------------
'W17A L
'------------------------
MOVL C00213 BC00213 V=500.0
SFTOF
MOVJ C00214 BC00214 VJ=20.00
MOVL C00215 BC00215 V=166.7 PL=0
REFP 3 C00216 BC00216
CALL JOB:SEARCH-R1
SET P0310 P0006
SFTON P0310
MOVL C00217 BC00217 V=166.7 PL=0
REFP 3 C00218 BC00218
CALL JOB:SEARCH-R1
SET P0310 P0006
SFTON P0310
MOVL C00219 BC00219 V=166.7 PL=0
SFTOF
'------------------------
'W17A P
'------------------------
SFTOF
MOVL C00220 BC00220 V=416.7
MOVL C00221 BC00221 V=166.7 PL=0
REFP 3 C00222 BC00222
CALL JOB:SEARCH-R1
SET P0311 P0006
SFTON P0311
MOVL C00223 BC00223 V=166.7 PL=0
REFP 3 C00224 BC00224
CALL JOB:SEARCH-R1
SET P0311 P0006
SFTON P0311
MOVL C00225 BC00225 V=166.7 PL=0
SFTOF
MOVJ C00226 BC00226 VJ=10.00
MOVJ C00227 BC00227 VJ=20.00
MOVJ C00228 BC00228 VJ=50.00
MOVJ C00229 BC00229 VJ=50.00
MOVJ C00230 BC00230 VJ=70.00
MOVJ C00231 BC00231 VJ=30.00
MOVJ C00232 BC00232 VJ=30.00
'------------------------
'------------------------
'LEWA STRONA PROFIL GORA
'------------------------
'------------------------
MOVJ C00233 BC00233 VJ=30.00
MOVJ C00234 BC00234 VJ=30.00
MOVJ C00235 BC00235 VJ=30.00
'------------------------
'W17B L
'------------------------
SFTOF
MOVJ C00236 BC00236 VJ=15.00
MOVL C00237 BC00237 V=166.7 PL=0
REFP 3 C00238 BC00238
CALL JOB:SEARCH-R1
SET P0350 P0006
SFTON P0350
MOVL C00239 BC00239 V=166.7 PL=0
REFP 3 C00240 BC00240
CALL JOB:SEARCH-R1
SET P0350 P0006
SFTON P0350
MOVL C00241 BC00241 V=166.7 PL=0
SFTOF
'------------------------
'W17B P
'------------------------
SFTOF
MOVL C00242 BC00242 V=333.3
MOVL C00243 BC00243 V=166.7 PL=0
REFP 3 C00244 BC00244
CALL JOB:SEARCH-R1
SET P0351 P0006
SFTON P0351
MOVL C00245 BC00245 V=166.7 PL=0
REFP 3 C00246 BC00246
CALL JOB:SEARCH-R1
SET P0351 P0006
SFTON P0351
MOVL C00247 BC00247 V=166.7 PL=0
SFTOF
'POPRAWID DOJAZD
'------------------------
'W15B L
'------------------------
SFTOF
MOVJ C00248 BC00248 VJ=10.00
MOVL C00249 BC00249 V=166.7 PL=0
REFP 3 C00250 BC00250
CALL JOB:SEARCH-R1
SET P0352 P0006
SFTON P0352
MOVL C00251 BC00251 V=166.7 PL=0
REFP 3 C00252 BC00252
CALL JOB:SEARCH-R1
SET P0352 P0006
SFTON P0352
MOVL C00253 BC00253 V=166.7 PL=0
SFTOF
'------------------------
'W15B P
'------------------------
SFTOF
MOVJ C00254 BC00254 VJ=20.00
MOVL C00255 BC00255 V=166.7 PL=0
REFP 3 C00256 BC00256
CALL JOB:SEARCH-R1
SET P0353 P0006
SFTON P0353
MOVL C00257 BC00257 V=166.7 PL=0
REFP 3 C00258 BC00258
CALL JOB:SEARCH-R1
SET P0353 P0006
SFTON P0353
MOVL C00259 BC00259 V=166.7 PL=0
SFTOF
'------------------------
'W18B L
'------------------------
SFTOF
MOVJ C00260 BC00260 VJ=50.00
MOVL C00261 BC00261 V=166.7 PL=0
REFP 3 C00262 BC00262
CALL JOB:SEARCH-R1
SET P0354 P0006
SFTON P0354
MOVL C00263 BC00263 V=166.7 PL=0
REFP 3 C00264 BC00264
CALL JOB:SEARCH-R1
SET P0354 P0006
SFTON P0354
MOVL C00265 BC00265 V=166.7 PL=0
SFTOF
'------------------------
'W18B P
'------------------------
SFTOF
MOVJ C00266 BC00266 VJ=50.00
MOVL C00267 BC00267 V=166.7 PL=0
REFP 3 C00268 BC00268
CALL JOB:SEARCH-R1
SET P0355 P0006
SFTON P0355
MOVL C00269 BC00269 V=166.7 PL=0
REFP 3 C00270 BC00270
CALL JOB:SEARCH-R1
SET P0355 P0006
SFTON P0355
MOVL C00271 BC00271 V=166.7 PL=0
SFTOF
'------------------------
'W13B L
'------------------------
SFTOF
MOVJ C00272 BC00272 VJ=50.00
MOVL C00273 BC00273 V=166.7 PL=0
REFP 3 C00274 BC00274
CALL JOB:SEARCH-R1
SET P0356 P0006
SFTON P0356
MOVL C00275 BC00275 V=166.7 PL=0
REFP 3 C00276 BC00276
CALL JOB:SEARCH-R1
SET P0356 P0006
SFTON P0356
MOVL C00277 BC00277 V=166.7 PL=0
SFTOF
'------------------------
'W13B P
'------------------------
SFTOF
MOVJ C00278 BC00278 VJ=50.00
MOVL C00279 BC00279 V=166.7 PL=0
REFP 3 C00280 BC00280
CALL JOB:SEARCH-R1
SET P0357 P0006
SFTON P0357
MOVL C00281 BC00281 V=166.7 PL=0
REFP 3 C00282 BC00282
CALL JOB:SEARCH-R1
SET P0357 P0006
SFTON P0357
MOVL C00283 BC00283 V=166.7 PL=0
SFTOF
'------------------------
'W19B L
'------------------------
SFTOF
MOVJ C00284 BC00284 VJ=50.00
MOVL C00285 BC00285 V=166.7 PL=0
REFP 3 C00286 BC00286
CALL JOB:SEARCH-R1
SET P0358 P0006
SFTON P0358
MOVL C00287 BC00287 V=166.7 PL=0
REFP 3 C00288 BC00288
CALL JOB:SEARCH-R1
SET P0358 P0006
SFTON P0358
MOVL C00289 BC00289 V=166.7 PL=0
SFTOF
'------------------------
'W19B P
'------------------------
SFTOF
MOVJ C00290 BC00290 VJ=50.00
MOVL C00291 BC00291 V=166.7 PL=0
REFP 3 C00292 BC00292
CALL JOB:SEARCH-R1
SET P0359 P0006
SFTON P0359
MOVL C00293 BC00293 V=166.7 PL=0
REFP 3 C00294 BC00294
CALL JOB:SEARCH-R1
SET P0359 P0006
SFTON P0359
MOVL C00295 BC00295 V=166.7 PL=0
SFTOF
'------------------------
'W14B L
'------------------------
SFTOF
MOVJ C00296 BC00296 VJ=50.00
MOVL C00297 BC00297 V=166.7 PL=0
REFP 3 C00298 BC00298
CALL JOB:SEARCH-R1
SET P0360 P0006
SFTON P0360
MOVL C00299 BC00299 V=166.7 PL=0
REFP 3 C00300 BC00300
CALL JOB:SEARCH-R1
SET P0360 P0006
SFTON P0360
MOVL C00301 BC00301 V=166.7 PL=0
SFTOF
'------------------------
'W14B P
'------------------------
SFTOF
MOVJ C00302 BC00302 VJ=50.00
MOVL C00303 BC00303 V=166.7 PL=0
REFP 3 C00304 BC00304
CALL JOB:SEARCH-R1
SET P0361 P0006
SFTON P0361
MOVL C00305 BC00305 V=166.7 PL=0
REFP 3 C00306 BC00306
CALL JOB:SEARCH-R1
SET P0361 P0006
SFTON P0361
MOVL C00307 BC00307 V=166.7 PL=0
SFTOF
MOVJ C00308 BC00308 VJ=50.00
MOVJ C00309 BC00309 VJ=50.00
MOVJ C00310 BC00310 VJ=50.00
MOVJ C00311 BC00311 VJ=50.00
'WELD
'WELD
'WELD
MOVJ C00312 BC00312 VJ=10.00
'**********************
'**********************
'POCZATEK SPAWANIA DOL
'**********************
'**********************
''
'**********************
'W1
'**********************
MOVJ C00313 BC00313 VJ=50.00
MOVJ C00314 BC00314 VJ=40.00
MOVL C00315 BC00315 V=166.7
SFTON P0104
MOVL C00316 BC00316 V=166.7
MACRO1 MJ#(0) ARGF14
ARCON
SFTON P0105
MOVL C00317 BC00317 V=11.7
ARCOF
SFTOF
MOVJ C00318 BC00318 VJ=20.00
MOVJ C00319 BC00319 VJ=30.00
MOVJ C00320 BC00320 VJ=50.00
MOVJ C00321 BC00321 VJ=40.00
MOVJ C00322 BC00322 VJ=20.00
'**********************
'W2
'**********************
SFTON P0108
MOVL C00323 BC00323 V=166.7
MACRO1 MJ#(0) ARGF9
ARCON
SFTON P0109
MOVL C00324 BC00324 V=11.7
MOVL C00325 BC00325 V=11.7
ARCOF
SFTOF
MOVL C00326 BC00326 V=333.3
MOVJ C00327 BC00327 VJ=40.00
MOVJ C00328 BC00328 VJ=70.00
MOVJ C00329 BC00329 VJ=20.00
MOVL C00330 BC00330 V=666.7
'**********************
'W3
'**********************
SFTON P0101
MACRO1 MJ#(0) ARGF9
MOVL C00331 BC00331 V=166.7
ARCON
SFTON P0100
MOVL C00332 BC00332 V=11.7
ARCOF
MOVL C00333 BC00333 V=166.7
SFTOF
MOVJ C00334 BC00334 VJ=30.00
MOVJ C00335 BC00335 VJ=30.00
MOVJ C00336 BC00336 VJ=50.00
MOVJ C00337 BC00337 VJ=30.00
MOVJ C00338 BC00338 VJ=40.00
'**********************
'W5
'**********************
MOVJ C00339 BC00339 VJ=50.00
MOVJ C00340 BC00340 VJ=25.00
MOVJ C00341 BC00341 VJ=30.00
'**********************
'W5
'**********************
MACRO1 MJ#(0) ARGF22
SFTON P0021
MOVL P0111 BP111 V=66.7
ARCON
WVON WEV#(2)
MOVL P0110 BP110 V=7.5
ARCOF
WVOF
SFTOF
MOVJ C00342 BC00342 VJ=20.00
MOVJ C00343 BC00343 VJ=20.00
'**********************
'W6
'**********************
MACRO1 MJ#(0) ARGF9
SFTON P0023
MOVL P0113 BP113 V=66.7
ARCON
WVON WEV#(2)
MOVL P0112 BP112 V=10.8
ARCOF
WVOF
SFTOF
MOVJ C00344 BC00344 VJ=10.00
MOVJ C00345 BC00345 VJ=30.00
MOVJ C00346 BC00346 VJ=30.00
MOVJ C00347 BC00347 VJ=40.00
MOVJ C00348 BC00348 VJ=40.00
MOVJ C00349 BC00349 VJ=40.00
MOVJ C00350 BC00350 VJ=40.00
MOVJ C00351 BC00351 VJ=20.00
MOVJ C00352 BC00352 VJ=10.00
MOVJ C00353 BC00353 VJ=20.00
MOVL C00354 BC00354 V=166.7
MACRO1 MJ#(0) ARGF14
MOVL C00355 BC00355 V=166.7
SFTON P0280
MOVL C00356 BC00356 V=166.7 PL=0
ARCON ASF#(22)
MOVL C00357 BC00357 V=9.2
MOVL C00358 BC00358 V=9.2
SFTON P0281
MOVL C00359 BC00359 V=9.2
MOVL C00360 BC00360 V=9.2
ARCOF
SFTOF
MOVL C00361 BC00361 V=250.0
MOVL C00362 BC00362 V=416.7
MOVJ C00363 BC00363 VJ=30.00
MOVJ C00364 BC00364 VJ=30.00
MOVJ C00365 BC00365 VJ=30.00
MOVJ C00366 BC00366 VJ=30.00
MOVJ C00367 BC00367 VJ=30.00
'7b
MOVL C00368 BC00368 V=333.3
MOVL C00369 BC00369 V=333.3
SFTON P0281
MOVL C00370 BC00370 V=166.7 PL=0
ARCON ASF#(22)
MOVL C00371 BC00371 V=9.2
MOVL C00372 BC00372 V=9.2
SFTON P0291
MOVL C00373 BC00373 V=9.2
MOVL C00374 BC00374 V=9.2
MOVL C00375 BC00375 V=9.2
ARCOF
SFTOF
'TUTAJ DODAC 7
'TUTAJ DODAC 7
'TUTAJ DODAC 7
MOVL C00376 BC00376 V=333.3
MOVL C00377 BC00377 V=333.3
MOVL C00378 BC00378 V=333.3
MOVJ C00379 BC00379 VJ=20.00
MOVJ C00380 BC00380 VJ=30.00
MOVJ C00381 BC00381 VJ=50.00
MOVJ C00382 BC00382 VJ=50.00
MOVJ C00383 BC00383 VJ=40.00
MOVJ C00384 BC00384 VJ=10.00
'**********************
'W9
'**********************
SFTON P0103
MACRO1 MJ#(0) ARGF9
MOVL C00385 BC00385 V=166.7
ARCON
SFTON P0102
MOVL C00386 BC00386 V=11.7
ARCOF
SFTOF
MOVL C00387 BC00387 V=166.7
'**********************
'SPOINA_PODLOGA_BRAK_ROZP
'**********************
MOVL C00388 BC00388 V=333.3
SFTON P0099
MOVL C00389 BC00389 V=166.7
ARCON
SFTON P0098
MOVL C00390 BC00390 V=11.7
ARCOF
MOVL C00391 BC00391 V=166.7
SFTOF
'SPOINA_PODLOGA_BRAK_ROZP
MOVJ C00392 BC00392 VJ=40.00
MOVJ C00393 BC00393 VJ=70.00
MOVJ C00394 BC00394 VJ=50.00
MOVJ C00395 BC00395 VJ=20.00
'**********************
'W10
'**********************
MOVL C00396 BC00396 V=333.3
SFTON P0106
MOVL C00397 BC00397 V=166.7
ARCON
SFTON P0107
MOVL C00398 BC00398 V=11.7
ARCOF
SFTOF
MOVL C00399 BC00399 V=333.3
MOVJ C00400 BC00400 VJ=50.00
'**********************
'**********************
'POCZATEK SPAWANIA BOKI
'**********************
'**********************
MOVJ C00401 BC00401 VJ=50.00
MOVJ C00402 BC00402 VJ=50.00
'**********************
'W13A
'**********************
SFTON P0305
MOVL C00403 BC00403 V=166.7 PL=0
SFTOF
MACRO1 MJ#(0) ARGF10
ARCON
SFTON P0304
MOVL C00404 BC00404 V=10.8
ARCOF
SFTOF
MOVL C00405 BC00405 V=250.0
'W13B
MOVJ C00406 BC00406 VJ=30.00
MOVJ C00407 BC00407 VJ=50.00
MOVL C00408 BC00408 V=500.0
'**********************
'W13B
'**********************
SFTON P0356
MOVL C00409 BC00409 V=133.3 PL=0
SFTOF
ARCON
SFTON P0357
MOVL C00410 BC00410 V=10.8
ARCOF
SFTOF
MOVL C00411 BC00411 V=250.0
MOVJ C00412 BC00412 VJ=30.00
MOVJ C00413 BC00413 VJ=40.00
MOVJ C00414 BC00414 VJ=30.00
MOVJ C00415 BC00415 VJ=30.00
'**********************
'W14A
'**********************
MOVL C00416 BC00416 V=250.0
SFTON P0301
MOVL C00417 BC00417 V=50.0 PL=0
SFTOF
ARCON
SFTON P0300
MOVL C00418 BC00418 V=10.8
MOVL C00419 BC00419 V=10.8
MOVL C00420 BC00420 V=10.8
ARCOF
SFTOF
MOVL C00421 BC00421 V=150.0
MOVJ C00422 BC00422 VJ=40.00
MOVJ C00423 BC00423 VJ=30.00
MOVJ C00424 BC00424 VJ=30.00
MOVJ C00425 BC00425 VJ=30.00
MOVJ C00426 BC00426 VJ=30.00
'**********************
'W14B
'**********************
SFTON P0360
MOVL C00427 BC00427 V=333.3
MOVL C00428 BC00428 V=133.3 PL=0
SFTOF
ARCON
SFTON P0361
MOVL C00429 BC00429 V=10.8
MOVL C00430 BC00430 V=10.8
MOVL C00431 BC00431 V=10.8
ARCOF
SFTOF
MOVL C00432 BC00432 V=166.7
MOVJ C00433 BC00433 VJ=40.00
MOVJ C00434 BC00434 VJ=40.00
MOVJ C00435 BC00435 VJ=30.00
MOVJ C00436 BC00436 VJ=40.00
MOVJ C00437 BC00437 VJ=30.00
MOVJ C00438 BC00438 VJ=30.00
MOVJ C00439 BC00439 VJ=30.00
MOVJ C00440 BC00440 VJ=30.00
MOVJ C00441 BC00441 VJ=30.00
'**********************
'W15A
'**********************
SFTON P0309
MOVL C00442 BC00442 V=66.7
MOVL C00443 BC00443 V=133.3 PL=0
SFTOF
ARCON
SFTON P0308
MOVL C00444 BC00444 V=10.8
ARCOF
SFTOF
MOVL C00445 BC00445 V=150.0
MOVJ C00446 BC00446 VJ=30.00
MOVJ C00447 BC00447 VJ=50.00
MOVJ C00448 BC00448 VJ=50.00
MOVJ C00449 BC00449 VJ=50.00
MOVJ C00450 BC00450 VJ=50.00
MOVJ C00451 BC00451 VJ=50.00
'**********************
'W15B
'**********************
SFTON P0352
MOVL C00452 BC00452 V=250.0
MOVL C00453 BC00453 V=83.3 PL=0
SFTOF
ARCON
SFTON P0353
MOVL C00454 BC00454 V=10.8
ARCOF
MOVL C00455 BC00455 V=66.7
SFTOF
MOVJ C00456 BC00456 VJ=40.00
MOVJ C00457 BC00457 VJ=50.00
MOVJ C00458 BC00458 VJ=50.00
'BRAK W TEJ DLUGOSCI
'**********************
'W16A
'**********************
'**********************
'W16B
'**********************
'BRAK W TEJ DLUGOSCI
'**********************
'W17A
'**********************
MOVJ C00459 BC00459 VJ=50.00
MOVJ C00460 BC00460 VJ=50.00
'**********************
'W17A
'**********************
SFTON P0310
MOVL C00461 BC00461 V=333.3
MOVL C00462 BC00462 V=166.7 PL=0
SFTOF
ARCON
SFTON P0311
MOVL C00463 BC00463 V=10.8
ARCOF
SFTOF
MOVL C00464 BC00464 V=333.3
MOVJ C00465 BC00465 VJ=30.00
MOVJ C00466 BC00466 VJ=30.00
MOVJ C00467 BC00467 VJ=50.00
MOVJ C00468 BC00468 VJ=50.00
MOVJ C00469 BC00469 VJ=50.00
MOVJ C00470 BC00470 VJ=50.00
MOVJ C00471 BC00471 VJ=50.00
MOVJ C00472 BC00472 VJ=30.00
MOVJ C00473 BC00473 VJ=30.00
'**********************
'W17B
'**********************
SFTON P0351
MOVL C00474 BC00474 V=166.7
MOVL C00475 BC00475 V=166.7 PL=0
SFTOF
ARCON
SFTON P0350
MOVL C00476 BC00476 V=10.8
ARCOF
SFTOF
MOVL C00477 BC00477 V=250.0
MOVJ C00478 BC00478 VJ=30.00
MOVJ C00479 BC00479 VJ=30.00
MOVJ C00480 BC00480 VJ=30.00
MOVJ C00481 BC00481 VJ=30.00
MOVJ C00482 BC00482 VJ=40.00
'**********************
'W18A
'**********************
SFTON P0306
MOVL C00483 BC00483 V=333.3
MOVL C00484 BC00484 V=166.7 PL=0
SFTOF
ARCON
SFTON P0307
MOVL C00485 BC00485 V=10.8
ARCOF
SFTOF
MOVL C00486 BC00486 V=250.0
MOVJ C00487 BC00487 VJ=30.00
MOVJ C00488 BC00488 VJ=30.00
MOVJ C00489 BC00489 VJ=50.00
MOVJ C00490 BC00490 VJ=50.00
MOVJ C00491 BC00491 VJ=50.00
'**********************
'W18B
'**********************
SFTON P0355
MOVL C00492 BC00492 V=166.7
MOVL C00493 BC00493 V=166.7 PL=0
SFTOF
ARCON
SFTON P0354
MOVL C00494 BC00494 V=10.8
ARCOF
MOVL C00495 BC00495 V=250.0
SFTOF
MOVJ C00496 BC00496 VJ=30.00
MOVJ C00497 BC00497 VJ=30.00
MOVJ C00498 BC00498 VJ=40.00
MOVJ C00499 BC00499 VJ=50.00
MOVJ C00500 BC00500 VJ=30.00
'**********************
'W19A
'**********************
MOVL C00501 BC00501 V=166.7
SFTON P0303
MOVL C00502 BC00502 V=166.7 PL=0
SFTOF
ARCON
SFTON P0302
MOVL C00503 BC00503 V=10.8
ARCOF
SFTOF
MOVL C00504 BC00504 V=150.0
MOVJ C00505 BC00505 VJ=30.00
MOVJ C00506 BC00506 VJ=50.00
MOVJ C00507 BC00507 VJ=50.00
'**********************
'W19B
'**********************
SFTON P0358
MOVL C00508 BC00508 V=500.0
MOVL C00509 BC00509 V=166.7 PL=0
SFTOF
ARCON
SFTON P0359
MOVL C00510 BC00510 V=10.8
ARCOF
SFTOF
MOVL C00511 BC00511 V=250.0
MOVJ C00512 BC00512 VJ=40.00
MOVJ C00513 BC00513 VJ=50.00
CALL JOB:MOVE_OUT_OF_TUNNEL
END
